PROGRAM P1_00_MAIN
VAR
END_VAR

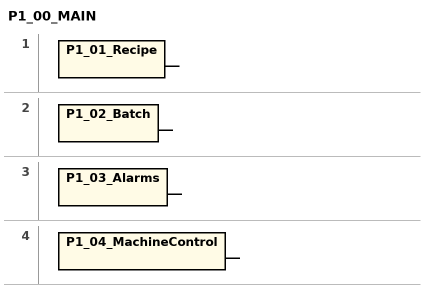
// NETWORK 1
P1_01_Recipe();

// NETWORK 2
P1_02_Batch();

// NETWORK 3
P1_03_Alarms();

// NETWORK 4
P1_04_MachineControl();

END_PROGRAM

(* stored: Version 1.1.0.1, ProductVersion 3.1.4026.13
   POU P1_00_MAIN: Id {283d4f7d-0013-4f57-a6c1-24d598d5c395}, SpecialFunc None *)
